// TwinCAT 3 PLC project Plc
// ProgramVersion: 3.1.4023.0
// libraries:
//   Tc2_Standard, * (Beckhoff Automation GmbH)
//   Tc2_System, * (Beckhoff Automation GmbH)
//   Tc3_Module, * (Beckhoff Automation GmbH)
// project tree:
//   / PlcTask.TcTTO (not stored)
//   DUTs/IO/PdoEntries/ Status_3D84275F.TcDUT, Ctrl_1EFB4D3B.TcDUT
//   DUTs/IO/PDOs/ InfoData_6F19DB2B.TcDUT (not stored), COM_ext_inputs_1F197B20.TcDUT, COM_ext_outputs_54D54ACC.TcDUT, WcState_9091E0EB.TcDUT, InfoData_32EB74EA.TcDUT, InfoData_E68C61CD.TcDUT (not stored), WcState_0B2B16F9.TcDUT (not stored), InfoData_2A97D6CF.TcDUT (not stored), Inputs_A65FACA4.TcDUT (not stored), Outputs_23C0ED1D.TcDUT (not stored)
//   DUTs/IO/Boxes/ EK1100_1FC0878B.TcDUT (not stored), EL6001_F578D623.TcDUT
//   DUTs/IO/Devices/ SyncUnitTask_2D604ED5.TcDUT (not stored), SyncUnitTasks_6FEB8257.TcDUT (not stored), SyncUnits_99E584AF.TcDUT (not stored)
//   DUTs/IO/Topology/ Term_1_EK1100_8210324B.TcDUT (not stored), Device_1_EtherCAT_6E94764C.TcDUT (not stored)
//   DUTs/IO/Base/ EtcSlaveBase_82538BE2.TcDUT (not stored), EtcSlaveBase_82538BE2.TcDUT (not stored), EtcSlaveBase_82538BE2.TcDUT (not stored), EtcSlaveTerminalBase_947E5A46.TcDUT (not stored), EtcSlaveBoxBase_77A0E4A7.TcDUT (not stored), EtcSlaveEndTerminalBase_866C7F0C.TcDUT (not stored), InputBase_8311D824.TcDUT (not stored), OutputBase_10CEE7DE.TcDUT (not stored), EtcMasterBase_62654B43.TcDUT (not stored)
//   GVLs/ GVL_iXlinker.TcGVL (not stored)
// real-time tasks:
//   TASK PlcTask: cycle T#10ms, priority 20, ADS port 350
// I/O:
//   DEVICE Device 1 (EtherCAT), AmsNetId 172.20.30.238.2.1
//     Term 1 (EK1100) [EK1100 EtherCAT Coupler (2A E-Bus)]
//       Term 2 (EL6001) [EL6001 Interface (RS232)]
// variable links:
//   Plc/Plc Instance <-> Device 1 (EtherCAT)/Term 1 (EK1100)
//     PlcTask Inputs/GVL_iXlinker.Device_1_EtherCAT.Term_1_EK1100.InfoData.State <-> InfoData/State
//   Plc/Plc Instance <-> Device 1 (EtherCAT)/Term 1 (EK1100)/Term 2 (EL6001)
//     PlcTask Inputs/GVL_iXlinker.Device_1_EtherCAT.Term_1_EK1100.Term_2_EL6001.COM_ext_inputs.Status/Transmit_accepted <-> COM ext. inputs/Status/Transmit accepted
//     PlcTask Inputs/GVL_iXlinker.Device_1_EtherCAT.Term_1_EK1100.Term_2_EL6001.COM_ext_inputs.Status/Receive_request <-> COM ext. inputs/Status/Receive request
//     PlcTask Inputs/GVL_iXlinker.Device_1_EtherCAT.Term_1_EK1100.Term_2_EL6001.COM_ext_inputs.Status/Init_accepted <-> COM ext. inputs/Status/Init accepted
//     PlcTask Inputs/GVL_iXlinker.Device_1_EtherCAT.Term_1_EK1100.Term_2_EL6001.COM_ext_inputs.Status/Buffer_full <-> COM ext. inputs/Status/Buffer full
//     PlcTask Inputs/GVL_iXlinker.Device_1_EtherCAT.Term_1_EK1100.Term_2_EL6001.COM_ext_inputs.Status/Parity_error <-> COM ext. inputs/Status/Parity error
//     PlcTask Inputs/GVL_iXlinker.Device_1_EtherCAT.Term_1_EK1100.Term_2_EL6001.COM_ext_inputs.Status/Framing_error <-> COM ext. inputs/Status/Framing error
//     PlcTask Inputs/GVL_iXlinker.Device_1_EtherCAT.Term_1_EK1100.Term_2_EL6001.COM_ext_inputs.Status/Overrun_error <-> COM ext. inputs/Status/Overrun error
//     PlcTask Inputs/GVL_iXlinker.Device_1_EtherCAT.Term_1_EK1100.Term_2_EL6001.COM_ext_inputs.Status/Input_length <-> COM ext. inputs/Status/Input length
//     PlcTask Inputs/GVL_iXlinker.Device_1_EtherCAT.Term_1_EK1100.Term_2_EL6001.COM_ext_inputs.Data_In[{0..49}] <-> COM ext. inputs/Data In {0..49}  (50 links)
//     PlcTask Outputs/GVL_iXlinker.Device_1_EtherCAT.Term_1_EK1100.Term_2_EL6001.COM_ext_outputs.Ctrl/Transmit_request <-> COM ext. outputs/Ctrl/Transmit request
//     PlcTask Outputs/GVL_iXlinker.Device_1_EtherCAT.Term_1_EK1100.Term_2_EL6001.COM_ext_outputs.Ctrl/Receive_accepted <-> COM ext. outputs/Ctrl/Receive accepted
//     PlcTask Outputs/GVL_iXlinker.Device_1_EtherCAT.Term_1_EK1100.Term_2_EL6001.COM_ext_outputs.Ctrl/Init_request <-> COM ext. outputs/Ctrl/Init request
//     PlcTask Outputs/GVL_iXlinker.Device_1_EtherCAT.Term_1_EK1100.Term_2_EL6001.COM_ext_outputs.Ctrl/Send_continuous <-> COM ext. outputs/Ctrl/Send continuous
//     PlcTask Outputs/GVL_iXlinker.Device_1_EtherCAT.Term_1_EK1100.Term_2_EL6001.COM_ext_outputs.Ctrl/Output_length <-> COM ext. outputs/Ctrl/Output length
//     PlcTask Outputs/GVL_iXlinker.Device_1_EtherCAT.Term_1_EK1100.Term_2_EL6001.COM_ext_outputs.Data_Out[{0..49}] <-> COM ext. outputs/Data Out {0..49}  (50 links)
//     PlcTask Inputs/GVL_iXlinker.Device_1_EtherCAT.Term_1_EK1100.Term_2_EL6001.WcState.WcState <-> WcState/WcState
//     PlcTask Inputs/GVL_iXlinker.Device_1_EtherCAT.Term_1_EK1100.Term_2_EL6001.WcState.InputToggle <-> WcState/InputToggle
//     PlcTask Inputs/GVL_iXlinker.Device_1_EtherCAT.Term_1_EK1100.Term_2_EL6001.InfoData.AdsAddr <-> InfoData/AdsAddr
//     PlcTask Inputs/GVL_iXlinker.Device_1_EtherCAT.Term_1_EK1100.Term_2_EL6001.InfoData.State <-> InfoData/State
//   Plc/Plc Instance <-> Device 1 (EtherCAT)
//     PlcTask Inputs/GVL_iXlinker.Device_1_EtherCAT.SyncUnits._default._unreferenced.WcState.WcState <-> SyncUnits/<default>/<unreferenced>/WcState/WcState
//     PlcTask Inputs/GVL_iXlinker.Device_1_EtherCAT.SyncUnits._default._unreferenced.InfoData.ObjectId <-> SyncUnits/<default>/<unreferenced>/InfoData/ObjectId
//     PlcTask Inputs/GVL_iXlinker.Device_1_EtherCAT.SyncUnits._default._unreferenced.InfoData.State <-> SyncUnits/<default>/<unreferenced>/InfoData/State
//     PlcTask Inputs/GVL_iXlinker.Device_1_EtherCAT.SyncUnits._default._unreferenced.InfoData.SlaveCount <-> SyncUnits/<default>/<unreferenced>/InfoData/SlaveCount
//     PlcTask Inputs/GVL_iXlinker.Device_1_EtherCAT.SyncUnits._default.PlcTask.WcState.WcState <-> SyncUnits/<default>/PlcTask/WcState/WcState
//     PlcTask Inputs/GVL_iXlinker.Device_1_EtherCAT.SyncUnits._default.PlcTask.InfoData.ObjectId <-> SyncUnits/<default>/PlcTask/InfoData/ObjectId
//     PlcTask Inputs/GVL_iXlinker.Device_1_EtherCAT.SyncUnits._default.PlcTask.InfoData.State <-> SyncUnits/<default>/PlcTask/InfoData/State
//     PlcTask Inputs/GVL_iXlinker.Device_1_EtherCAT.SyncUnits._default.PlcTask.InfoData.SlaveCount <-> SyncUnits/<default>/PlcTask/InfoData/SlaveCount
//     PlcTask Inputs/GVL_iXlinker.Device_1_EtherCAT.Inputs.SlaveCount <-> Inputs/SlaveCount
//     PlcTask Inputs/GVL_iXlinker.Device_1_EtherCAT.Inputs.DevState <-> Inputs/DevState
//     PlcTask Inputs/GVL_iXlinker.Device_1_EtherCAT.Inputs.Frm0State <-> Inputs/Frm0State
//     PlcTask Inputs/GVL_iXlinker.Device_1_EtherCAT.Inputs.Frm0WcState <-> Inputs/Frm0WcState
//     PlcTask Inputs/GVL_iXlinker.Device_1_EtherCAT.Inputs.Frm0InputToggle <-> Inputs/Frm0InputToggle
//     PlcTask Outputs/GVL_iXlinker.Device_1_EtherCAT.Outputs.DevCtrl <-> Outputs/DevCtrl
//     PlcTask Outputs/GVL_iXlinker.Device_1_EtherCAT.Outputs.Frm0Ctrl <-> Outputs/Frm0Ctrl
//     PlcTask Outputs/GVL_iXlinker.Device_1_EtherCAT.Outputs.Frm0WcCtrl <-> Outputs/Frm0WcCtrl
//     PlcTask Inputs/GVL_iXlinker.Device_1_EtherCAT.InfoData.ChangeCount <-> InfoData/ChangeCount
//     PlcTask Inputs/GVL_iXlinker.Device_1_EtherCAT.InfoData.DevId <-> InfoData/DevId
//     PlcTask Inputs/GVL_iXlinker.Device_1_EtherCAT.InfoData.AmsNetId <-> InfoData/AmsNetId
//     PlcTask Inputs/GVL_iXlinker.Device_1_EtherCAT.InfoData.CfgSlaveCount <-> InfoData/CfgSlaveCount
//     PlcTask Inputs/GVL_iXlinker.Device_1_EtherCAT.InfoData.DcToTcTimeOffset <-> InfoData/DcToTcTimeOffset
//     PlcTask Inputs/GVL_iXlinker.Device_1_EtherCAT.InfoData.DcToExtTimeOffset <-> InfoData/DcToExtTimeOffset

// ---- DUTs/IO/PdoEntries/Status_3D84275F.TcDUT
{attribute 'GeneratedUsingTerminal: EL6001-0000-0020'}
{attribute addProperty BoxType "EL6001-0000-0020"}
{attribute addProperty Id "Transmit_acceptedBOOL1Receive_requestBOOL1Init_acceptedBOOL1Buffer_fullBOOL1Parity_errorBOOL1Framing_errorBOOL1Overrun_errorBOOL1Input_lengthUSINT1"}
{attribute addProperty CRC "1032071007"}
{attribute addProperty Size "8"}
TYPE Status_3D84275F :
STRUCT
	{attribute addProperty Name "Transmit_accepted"}
	Transmit_accepted : BOOL;
	{attribute addProperty Name "Receive_request"}
	Receive_request : BOOL;
	{attribute addProperty Name "Init_accepted"}
	Init_accepted : BOOL;
	{attribute addProperty Name "Buffer_full"}
	Buffer_full : BOOL;
	{attribute addProperty Name "Parity_error"}
	Parity_error : BOOL;
	{attribute addProperty Name "Framing_error"}
	Framing_error : BOOL;
	{attribute addProperty Name "Overrun_error"}
	Overrun_error : BOOL;
	{attribute addProperty Name "Input_length"}
	Input_length : USINT;
END_STRUCT
END_TYPE

// ---- DUTs/IO/PdoEntries/Ctrl_1EFB4D3B.TcDUT
{attribute 'GeneratedUsingTerminal: EL6001-0000-0020'}
{attribute addProperty BoxType "EL6001-0000-0020"}
{attribute addProperty Id "Transmit_requestBOOL1Receive_acceptedBOOL1Init_requestBOOL1Send_continuousBOOL1Output_lengthUSINT1"}
{attribute addProperty CRC "519785787"}
{attribute addProperty Size "5"}
TYPE Ctrl_1EFB4D3B :
STRUCT
	{attribute addProperty Name "Transmit_request"}
	Transmit_request : BOOL;
	{attribute addProperty Name "Receive_accepted"}
	Receive_accepted : BOOL;
	{attribute addProperty Name "Init_request"}
	Init_request : BOOL;
	{attribute addProperty Name "Send_continuous"}
	Send_continuous : BOOL;
	{attribute addProperty Name "Output_length"}
	Output_length : USINT;
END_STRUCT
END_TYPE

// ---- DUTs/IO/PDOs/COM_ext_inputs_1F197B20.TcDUT
{attribute 'GeneratedUsingTerminal: EL6001-0000-0020'}
{attribute addProperty BoxType "EL6001-0000-0020"}
{attribute addProperty Id "StatusAT %I*Status_3D84275F8Data_InAT %I*ARRAY[0..49] OF UINT100"}
{attribute addProperty CRC "1924718055"}
{attribute addProperty Size "108"}
TYPE COM_ext_inputs_1F197B20 EXTENDS InputBase_8311D824 :
STRUCT
	{attribute addProperty Name "Status"}
	Status AT %I* : Status_3D84275F;
	{attribute addProperty Name "Data_In"}
	Data_In AT %I* : ARRAY[0..49] OF UINT;
END_STRUCT
END_TYPE

// ---- DUTs/IO/PDOs/COM_ext_outputs_54D54ACC.TcDUT
{attribute 'GeneratedUsingTerminal: EL6001-0000-0020'}
{attribute addProperty BoxType "EL6001-0000-0020"}
{attribute addProperty Id "CtrlAT %Q*Ctrl_1EFB4D3B5Data_OutAT %Q*ARRAY[0..49] OF UINT100"}
{attribute addProperty CRC "3984205705"}
{attribute addProperty Size "105"}
TYPE COM_ext_outputs_54D54ACC EXTENDS OutputBase_10CEE7DE :
STRUCT
	{attribute addProperty Name "Ctrl"}
	Ctrl AT %Q* : Ctrl_1EFB4D3B;
	{attribute addProperty Name "Data_Out"}
	Data_Out AT %Q* : ARRAY[0..49] OF UINT;
END_STRUCT
END_TYPE

// ---- DUTs/IO/PDOs/WcState_9091E0EB.TcDUT
{attribute 'GeneratedUsingTerminal: EL6001-0000-0020'}
{attribute addProperty BoxType "EL6001-0000-0020"}
{attribute addProperty Id "WcStateAT %I*BOOL1InputToggleAT %I*BOOL1"}
{attribute addProperty CRC "2425479403"}
{attribute addProperty Size "2"}
TYPE WcState_9091E0EB :
STRUCT
	{attribute addProperty Name "WcState"}
	WcState AT %I* : BOOL;
	{attribute addProperty Name "InputToggle"}
	InputToggle AT %I* : BOOL;
END_STRUCT
END_TYPE

// ---- DUTs/IO/PDOs/InfoData_32EB74EA.TcDUT
{attribute 'GeneratedUsingTerminal: EL6001-0000-0020'}
{attribute addProperty BoxType "EL6001-0000-0020"}
{attribute addProperty Id "AdsAddrAT %I*AMSADDR8StateAT %I*UINT2"}
{attribute addProperty CRC "854291690"}
{attribute addProperty Size "10"}
TYPE InfoData_32EB74EA EXTENDS InputBase_8311D824 :
STRUCT
	{attribute addProperty Name "AdsAddr"}
	AdsAddr AT %I* : AMSADDR;
	{attribute addProperty Name "State"}
	State AT %I* : UINT;
END_STRUCT
END_TYPE

// ---- DUTs/IO/Boxes/EL6001_F578D623.TcDUT
{attribute 'GeneratedUsingTerminal: EL6001-0000-0020'}
{attribute addProperty BoxType "EL6001-0000-0020"}
{attribute addProperty Description "EL6001 Interface (RS232)"}
{attribute addProperty Physics "KK"}
{attribute addProperty Id "COM_ext_inputsAT %I*COM_ext_inputs_1F197B20108COM_ext_outputsAT %Q*COM_ext_outputs_54D54ACC105WcStateAT %I*WcState_9091E0EB2InfoDataAT %I*InfoData_32EB74EA10"}
{attribute addProperty CRC "4118337059"}
{attribute addProperty Size "225"}
TYPE EL6001_F578D623 EXTENDS EtcSlaveTerminalBase_947E5A46 :
STRUCT
	{attribute addProperty Name "COM_ext_inputs"}
	COM_ext_inputs : COM_ext_inputs_1F197B20;
	{attribute addProperty Name "COM_ext_outputs"}
	COM_ext_outputs : COM_ext_outputs_54D54ACC;
	{attribute addProperty Name "WcState"}
	WcState : WcState_9091E0EB;
	{attribute addProperty Name "InfoData"}
	InfoData : InfoData_32EB74EA;
END_STRUCT
END_TYPE
